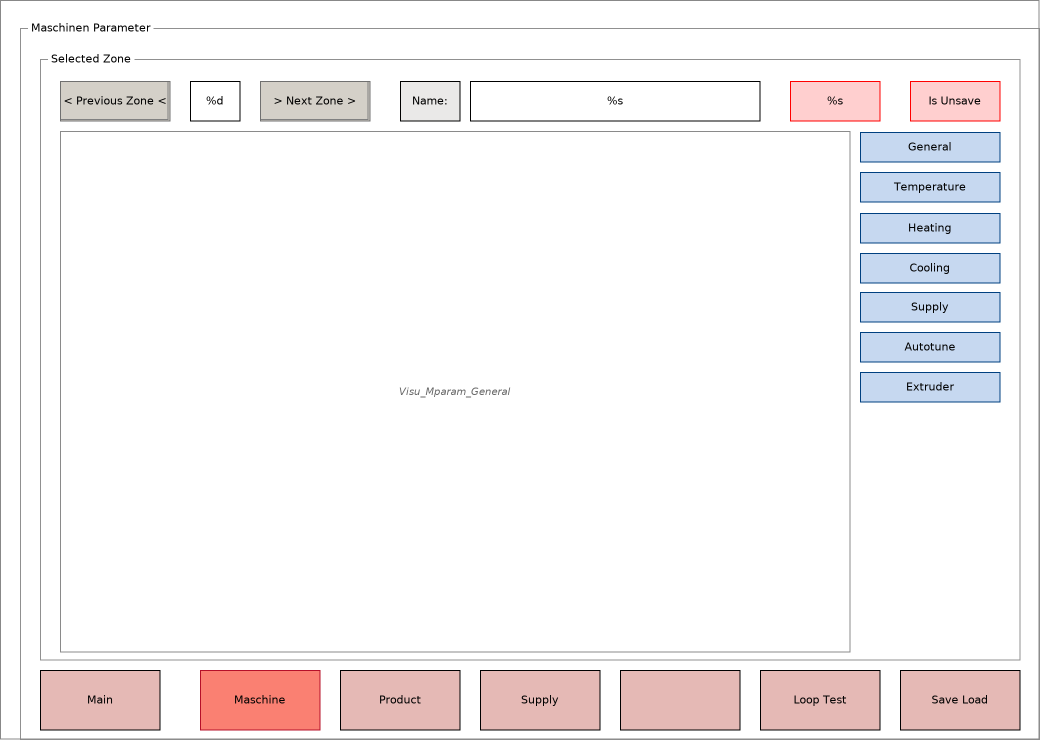
VISUALIZATION Visu_MParam  // 1040x740
    GroupBox (20,20 1020x720), "Maschinen Parameter"
        Rectangle (20,650 120x60), "Main"
            OnMouseClick: change screen: Visu_Main
        Rectangle (880,650 120x60), "Save Load"
            OnMouseClick: change screen: Visu_SaveLoad
        Rectangle (320,650 120x60), "Product"
            OnMouseClick: change screen: Visu_PParam
        Rectangle (180,650 120x60), "Maschine"
            OnMouseClick: change screen: Visu_MParam
        Rectangle (460,650 120x60), "Supply"
            OnMouseClick: change screen: Visu_Supply
        Rectangle (600,650 120x60)
        GroupBox (20,31 980x609), "Selected Zone"
            Rectangle (150,30 50x40), "%d", text variable: nVisuCount
            Button (20,30 110x40), "< Previous Zone <"
                tap bVisuBefore
            Button (220,30 110x40), "> Next Zone >"
                tap bVisuNext
            Rectangle (750,30 90x40), "%s", text variable: stMParam_Visu.sInUse, colour toggle: aaaPfwTempMparamFromHmi[nVisuCount].InUse
                OnMouseClick: toggle aaaPfwTempMparamFromHmi[nVisuCount].InUse
                OnMouseClick: execute { stParamsUnsave.mParams[nVisuCount]:=TRUE; }
            Rectangle (430,30 290x40), "%s", text variable: aaaPfwTempMparamFromHmi[nVisuCount].ZoneName
                OnMouseClick: write the text variable via Edit
                OnMouseClick: execute { stParamsUnsave.mParams[nVisuCount]:=TRUE; }
            Rectangle (360,30 60x40), "Name:"
            Rectangle (870,30 90x40), "Is Unsave", invisible if: Not stParamsUnsave.mParams[nVisuCount]
                OnMouseClick: execute { aaaPfwTempMparamFromHmi[nVisuCount].SaveDelay:=1000; stParamsUnsave.mParams[nVisuCount]:=FALSE; }
            Rectangle (820,81 140x30), "General", colour toggle: stMParam_Visu.nActiveParamList=0
                OnMouseClick: execute { stMParam_Visu.nActiveParamList:=0; }
            Frame (20,80 790x521), frame switch variable: stMParam_Visu.nActiveParamList
                shows Visu_Mparam_General()
                shows Visu_Mparam_Temperature()
                shows Visu_Mparam_Heat()
                shows Visu_Mparam_Cool()
                shows Visu_Mparam_Supply()
                shows Visu_Mparam_Autotune()
                shows Visu_Mparam_Extruder()
            Rectangle (820,202 140x30), "Cooling", colour toggle: stMParam_Visu.nActiveParamList=3
                OnMouseClick: execute { stMParam_Visu.nActiveParamList:=3; }
            Rectangle (820,162 140x30), "Heating", colour toggle: stMParam_Visu.nActiveParamList=2
                OnMouseClick: execute { stMParam_Visu.nActiveParamList:=2; }
            Rectangle (820,321 140x30), "Extruder", colour toggle: stMParam_Visu.nActiveParamList=6, invisible if: NOT MAIN.bFirstCycle
                OnMouseClick: execute { stMParam_Visu.nActiveParamList:=6; }
            Rectangle (820,281 140x30), "Autotune", colour toggle: stMParam_Visu.nActiveParamList=5
                OnMouseClick: execute { stMParam_Visu.nActiveParamList:=5; }
            Rectangle (820,241 140x30), "Supply", colour toggle: stMParam_Visu.nActiveParamList=4
                OnMouseClick: execute { stMParam_Visu.nActiveParamList:=4; }
            Rectangle (820,121 140x30), "Temperature", colour toggle: stMParam_Visu.nActiveParamList=1
                OnMouseClick: execute { stMParam_Visu.nActiveParamList:=1; }
        Rectangle (740,650 120x60), "Loop Test"
            OnMouseClick: change screen: Visu_LoopTest
END_VISUALIZATION

(* stored: Version 1.1.0.1
   Visu Visu_MParam: Id {7114911d-3688-48ce-b2a3-d7acdb234f55} *)
